			R3.Reamer[1](
				(*FB Inputs*)
					Enable_Motion:= All_Estops_OK,
					Fronius_Ream:= TRUE,
                    Binzel_Ream:= FALSE,  (*optional*)
					
					Ream_REQ:= R3.Peripheral_Req.1 AND ((R3.Task_ID_Ack=Tip_Dress)OR (R3.In_T1 AND R3.Peripheral_Req.5)),
					Ream_Time:= T#2S,
					Ream_Clamp_Open:= R3.Reamer[1].N01.I.1,
					Spray_REQ:= R3.Peripheral_Req.2 AND ((R3.Task_ID_Ack=Tip_Dress)OR (R3.In_T1 AND R3.Peripheral_Req.5)),
					Spray_Time:= T#2S,
					F_WireCutter_REQ:= R3.Peripheral_Req.4 AND ((R3.Task_ID_Ack=Tip_Dress)OR (R3.In_T1 AND R3.Peripheral_Req.5)),
					F_WireCutter_Time:= T#1S,
					
				(*FB Outputs*)
					Reaming_Complete=> ,(*mapped in cell services*)
					(*The following are for Binzel type reamers only*)
					LifterUp_ACK=> , (*mapped in cell services*)
					Clamp_ACK=>,(*mapped in cell services*)
					Injector_ACK=> ,(*mapped in cell services*)
					WireCutter_ACK=> (*mapped in cell services*)
					);
			
			(*R3.Reamer[1](
				(*FB Inputs*)
					Enable_Motion:= All_Estops_OK,
					Fronius_Ream:= TRUE,
                    Binzel_Ream:= FALSE,  (*optional*)
					Ream_REQ:= R3.Peripheral_Req.5 AND (R3.Task_ID_Ack=Tip_Dress),

				(*FB Outputs*)
					Reaming_Complete=> ,(*mapped in cell services*)
					);*)
		(*Call Actual Object*)
		R3();
		(*Output Data*)
		Out_To_ICxx.Robot[3].Robot_Type:= R3.FB_In.Robot_Type;
		Out_To_ICxx.Robot[3].Status:= R3.Status;
		Out_To_ICxx.Robot[3].Axis_Data[1]:= R3.S_Axis_Pos_Raw;
		Out_To_ICxx.Robot[3].In_Image:= R3.Input_Image;
		Out_To_ICxx.Robot[3].Out_Image:= R3.Output_Image;
		Out_To_ICxx.Robot[3].Discrete_ImageFSOE:= R3.Discrete_Image_FSoE;
		Out_To_ICxx.Robot[3].Options:= R3.FB_In.Options;
			Out_To_ICxx.Robot[3].WS_Discrete_Image[1]:= R3.WS[1].Discrete_Image;
			Out_To_ICxx.Robot[3].WS_Discrete_Image[2]:= R3.WS[2].Discrete_Image;
 			Out_To_ICxx.Robot[3].ATI_Discrete_Image:= R3.ATI[1].Discrete_Image;
			Out_To_ICxx.Robot[3].Reamer_Discrete_Image:= R3.Reamer[1].Discrete_Image;
			Out_To_ICxx.Robot[3].Fronius_Status:= R3.Fronius_Status;
		Out_To_ICxx.Robot[3].Ped_IO_ToShow[1]:= 0;			(*Set to Ped value if this robots ecat string contains the Ped's IO*)
		Out_To_ICxx.Robot[3].Ped_IO_ToShow[2]:= 0;			(*Set to Ped value if this robots ecat string contains the Ped's IO*)
		Out_To_ICxx.Robot[3].ECAT_Cable_Breaks:= R3.ECatSlave_Cable_Breaks;
		Out_To_ICxx.Robot[3].CT:= R3.CT;


(*R4 ------------------------*)
		(*Input Data*)
		R4.FB_In.Robot_Type:=KUKA_KRC4_SAFEOP;
		R4.FB_In.Install_Zero_Orientation:= 0; 	(*Set this value between 0 and 359 to set the zero position of the robot physical install with reference to 12 o'clock symbol on UI screens*)
		R4.FB_In.Under_Construction:= GTAC_CONFIG.Under_Construction;
		R4.FB_In.In_SIM_Mode:= GTAC_CONFIG.In_SIM_Mode;
		R4.FB_In.SIM_StartWorkAround:= FALSE;  (*Main.SIM_WorkAround_StartRobots*)
		R4.FB_In.CoE_Read_Trigger:= (GTAC_CONFIG.Option_Robot_Count>=4) AND Pulse_CoERead;
		R4.FB_In.Ecat_Master_AmsNetID:= MAIN.ECAT_Master.AmsID;
		R4.FB_In.Prev_EcatNode_Present:= NOT R3.EK1100_NotPresent; (*Ensure Previous Node Exists to determine Ecat Cable Break of this Devices Input Cable*)
		R4.FB_In.Safety_RST:=SAFETY_RESET;
		R4.FB_In.Enable_Motion:= All_Estops_OK OR GTAC_CONFIG.Under_Construction;
		R4.FB_In.Alarm_RST:=In_From_ICxx.ControlPower1;
		R4.FB_In.Select_Play:=FALSE;
		R4.FB_In.Select_Teach:=FALSE;
		R4.FB_In.Select_Remote:=FALSE;
		R4.FB_In.Start_Scan:=In_From_ICxx.StartRobots;
		R4.FB_In.Stop_Scan:=In_From_ICxx.StopRobots;
		R4.FB_In.Stop_Scan2:=FALSE;
		R4.FB_In.In_DryCycle:= GTAC_CONFIG.Dry_Cycle_Enabled;
		R4.FB_In.Low_Speed:= GTAC_CONFIG.Low_Speed_Enabled;
		R4.FB_In.Speed_Request:= In_From_ICxx.Global_Robot_Speed;
		R4.FB_In.Force_MasterTest_Req:= Cell_Services_Prog.Human_Reqs_MasterTest OR Cell_Services_Prog.A_Robot_Reqs_MasterTest;
		R4.FB_In.Force_BrakeTest_Req:= Cell_Services_Prog.Human_Reqs_BrakeTest OR Cell_Services_Prog.A_Robot_Reqs_BrakeTest;
		R4.FB_In.Major_Faults:= Faults.System_Major_Fault;
		R4.FB_In.Teach_Interlock:=R4_Data.Teach_Interlock;
		R4.FB_In.Weld_Inhibit:=In_From_ICxx.Rxx_Weld_Inhibit;
		R4.FB_In.Option_Disable_WaterFLT:= FALSE AND GTAC_CONFIG.Under_Construction OR (MAIN.R4.Task_ID_Ack=Tip_Change_EXT); (*Used to disable water fault if no water is present. use with caution*)
		R4.FB_In.OK_ToEnter_EquipInterf1:=R4_Data.OK_ToEnter_EquipInterf1;
		R4.FB_In.OK_ToEnter_EquipInterf2:=R4_Data.OK_ToEnter_EquipInterf2;
		R4.FB_In.OK_ToEnter_EquipInterf3:=R4_Data.OK_ToEnter_EquipInterf3;
		R4.FB_In.OK_ToEnter_EquipInterf4:=R4_Data.OK_ToEnter_EquipInterf4;
		R4.FB_In.OK_ToEnter_EquipInterf5:=R4_Data.OK_ToEnter_EquipInterf5;
		R4.FB_In.OK_ToEnter_EquipInterf6:=R4_Data.OK_ToEnter_EquipInterf6;
		R4.FB_In.OK_ToEnter_EquipInterf7:=R4_Data.OK_ToEnter_EquipInterf7;
		R4.FB_In.OK_ToEnter_EquipInterf8:=R4_Data.OK_ToEnter_EquipInterf8;
		R4.FB_In.OK_ToEnter_EquipInterf9:=R4_Data.OK_ToEnter_EquipInterf9;
		R4.FB_In.OK_ToEnter_HumanInterf1:=R4_Data.OK_ToEnter_HumanInterf1;
		R4.FB_In.OK_ToEnter_HumanInterf2:=R4_Data.OK_ToEnter_HumanInterf2;
		R4.FB_In.OK_ToEnter_HumanInterf3:=R4_Data.OK_ToEnter_HumanInterf3;
		R4.FB_In.OK_ToEnter_HumanInterf4:=R4_Data.OK_ToEnter_HumanInterf4;
		R4.FB_In.OK_ToEnter_HumanInterf5:=R4_Data.OK_ToEnter_HumanInterf5;
		R4.FB_In.OK_ToEnter_HumanInterf6:=R4_Data.OK_ToEnter_HumanInterf6;
		R4.FB_In.OK_ToEnter_HumanInterf7:=R4_Data.OK_ToEnter_HumanInterf7;
		R4.FB_In.OK_ToEnter_RobotInterfs:= R4_Data.OK_ToEnter_RobotInterfs;
		R4.FB_In.Fix_ID:=R4_Data.Fix_ID[R4.Location_Index];
		R4.FB_In.Model_ID:=R4_Data.Model_ID[R4.Location_Index];
		R4.FB_In.Task_ID:=R4_Data.Task_ID[R4.Location_Index];
		R4.FB_In.Proceed_From_Pounce:=R4_Data.Proceed_From_Pounce[R4.Location_Index];
		R4.FB_In.Complete_Ack:=R4_Data.Complete_Ack[R4.Location_Index];
		R4.FB_In.PeripheralReq_Ack:=R4_Data.PeripheralReq_Ack[R4.Location_Index];
		R4.FB_In.AuxReq_Ack:=R4_Data.AuxReq_Ack[R4.Location_Index];
		R4.FB_In.User_Inputs.0:= FALSE;
		R4.FB_In.User_Inputs.1:= FALSE;
		R4.FB_In.User_Inputs.2:= FALSE;
		R4.FB_In.User_Inputs.3:= FALSE;
		R4.FB_In.User_Inputs.4:= FALSE;
		R4.FB_In.User_Inputs.5:= FALSE;
		R4.FB_In.User_Inputs.6:= FALSE;
		R4.FB_In.User_Inputs.7:= FALSE;
			(*Configure Options Amounts*)
			R4.FB_In.Options.WeldCont_Amount:=0; 					(*Select amount of Spot Type Weld Controllers here (0 min, 4 max)*)
			R4.FB_In.Options.WaterStand_Amount:= 0;				(*Select amount of Water Stands here (0 min, 2 max)*)
			R4.FB_In.Options.MIGCont_Amount:= 0;					(*Select amount of MIG Type Weld Controllers here (0 min, 1 max)*)
			R4.FB_In.Options.Reamer_Amount:= 0;					(*Select amount of Tip Reamers here (0 min, 1 max)*)
			R4.FB_In.Options.EOAT_Amount:= 1;						(*Assign EOAT number to robot (0 min, 10 max)*)
			(*Configure Options Parameters*)

		(*Call Actual Object*)
		R4();
		(*Output Data*)
		Out_To_ICxx.Robot[4].Robot_Type:= R4.FB_In.Robot_Type;
		Out_To_ICxx.Robot[4].Status:= R4.Status;
		Out_To_ICxx.Robot[4].Axis_Data[1]:= R4.S_Axis_Pos_Raw;
		Out_To_ICxx.Robot[4].Axis_Data[7]:= R4.External_Axis_Pos_Raw; (*Actual value coming from robot*)
		Out_To_ICxx.Robot[4].In_Image:= R4.Input_Image;
		Out_To_ICxx.Robot[4].Out_Image:= R4.Output_Image;
		Out_To_ICxx.Robot[4].Discrete_ImageFSOE:= R4.Discrete_Image_FSoE;
		Out_To_ICxx.Robot[4].Options:= R4.FB_In.Options;
			Out_To_ICxx.Robot[4].WS_Discrete_Image[1]:= R4.WS[1].Discrete_Image;
			Out_To_ICxx.Robot[4].WS_Discrete_Image[2]:= R4.WS[2].Discrete_Image;
 			Out_To_ICxx.Robot[4].ATI_Discrete_Image:= R4.ATI[1].Discrete_Image;
			Out_To_ICxx.Robot[4].Reamer_Discrete_Image:= R4.Reamer[1].Discrete_Image;
			Out_To_ICxx.Robot[4].Fronius_Status:= R4.Fronius_Status;
		Out_To_ICxx.Robot[4].Ped_IO_ToShow[1]:= 0;			(*Set to Ped value if this robots ecat string contains the Ped's IO*)
		Out_To_ICxx.Robot[4].Ped_IO_ToShow[2]:= 0;			(*Set to Ped value if this robots ecat string contains the Ped's IO*)
		Out_To_ICxx.Robot[4].ECAT_Cable_Breaks:= R4.ECatSlave_Cable_Breaks;
		Out_To_ICxx.Robot[4].CT:= R4.CT;



(*R5 ------------------------*)
		(*Input Data*)
		R5.FB_In.Robot_Type:=KUKA_KRC4_SAFEOP_Turntable;
		R5.FB_In.Install_Zero_Orientation:= 0; 	(*Set this value between 0 and 359 to set the zero position of the robot physical install with reference to 12 o'clock symbol on UI screens*)
		R5.FB_In.Under_Construction:= GTAC_CONFIG.Under_Construction;
		R5.FB_In.In_SIM_Mode:= GTAC_CONFIG.In_SIM_Mode;
		R5.FB_In.SIM_StartWorkAround:= FALSE;  (*Main.SIM_WorkAround_StartRobots*)
		R5.FB_In.CoE_Read_Trigger:= (GTAC_CONFIG.Option_Robot_Count>=5) AND Pulse_CoERead;
		R5.FB_In.Ecat_Master_AmsNetID:= MAIN.ECAT_Master.AmsID;
		R5.FB_In.Prev_EcatNode_Present:= NOT R4.EK1100_NotPresent; (*Ensure Previous Node Exists to determine Ecat Cable Break of this Devices Input Cable*)
		R5.FB_In.Safety_RST:=SAFETY_RESET;
		R5.FB_In.Enable_Motion:= All_Estops_OK OR GTAC_CONFIG.Under_Construction;
		R5.FB_In.Alarm_RST:=In_From_ICxx.ControlPower1;
		R5.FB_In.Select_Play:=FALSE;
		R5.FB_In.Select_Teach:=FALSE;
		R5.FB_In.Select_Remote:=FALSE;
		R5.FB_In.Start_Scan:=In_From_ICxx.StartRobots;
		R5.FB_In.Stop_Scan:=In_From_ICxx.StopRobots;
		R5.FB_In.Stop_Scan2:=FALSE;
		R5.FB_In.In_DryCycle:= GTAC_CONFIG.Dry_Cycle_Enabled;
		R5.FB_In.Low_Speed:= GTAC_CONFIG.Low_Speed_Enabled;
		R5.FB_In.Speed_Request:= In_From_ICxx.Global_Robot_Speed;
		R5.FB_In.Force_MasterTest_Req:= Cell_Services_Prog.Human_Reqs_MasterTest OR Cell_Services_Prog.A_Robot_Reqs_MasterTest;
		R5.FB_In.Force_BrakeTest_Req:= Cell_Services_Prog.Human_Reqs_BrakeTest OR Cell_Services_Prog.A_Robot_Reqs_BrakeTest;
		R5.FB_In.Major_Faults:= Faults.System_Major_Fault;
		R5.FB_In.Teach_Interlock:=R5_Data.Teach_Interlock;
		R5.FB_In.Weld_Inhibit:=In_From_ICxx.Rxx_Weld_Inhibit;
		R5.FB_In.Option_Disable_WaterFLT:= FALSE AND GTAC_CONFIG.Under_Construction OR (MAIN.R5.Task_ID_Ack=Tip_Change_EXT); (*Used to disable water fault if no water is present. use with caution*)
		R5.FB_In.OK_ToEnter_EquipInterf1:=R5_Data.OK_ToEnter_EquipInterf1;
		R5.FB_In.OK_ToEnter_EquipInterf2:=R5_Data.OK_ToEnter_EquipInterf2;
		R5.FB_In.OK_ToEnter_EquipInterf3:=R5_Data.OK_ToEnter_EquipInterf3;
		R5.FB_In.OK_ToEnter_EquipInterf4:=R5_Data.OK_ToEnter_EquipInterf4;
		R5.FB_In.OK_ToEnter_EquipInterf5:=R5_Data.OK_ToEnter_EquipInterf5;
		R5.FB_In.OK_ToEnter_EquipInterf6:=R5_Data.OK_ToEnter_EquipInterf6;
		R5.FB_In.OK_ToEnter_EquipInterf7:=R5_Data.OK_ToEnter_EquipInterf7;
		R5.FB_In.OK_ToEnter_EquipInterf8:=R5_Data.OK_ToEnter_EquipInterf8;
		R5.FB_In.OK_ToEnter_EquipInterf9:=R5_Data.OK_ToEnter_EquipInterf9;
		R5.FB_In.OK_ToEnter_HumanInterf1:=R5_Data.OK_ToEnter_HumanInterf1;
		R5.FB_In.OK_ToEnter_HumanInterf2:=R5_Data.OK_ToEnter_HumanInterf2;
		R5.FB_In.OK_ToEnter_HumanInterf3:=R5_Data.OK_ToEnter_HumanInterf3;
		R5.FB_In.OK_ToEnter_HumanInterf4:=R5_Data.OK_ToEnter_HumanInterf4;
		R5.FB_In.OK_ToEnter_HumanInterf5:=R5_Data.OK_ToEnter_HumanInterf5;
		R5.FB_In.OK_ToEnter_HumanInterf6:=R5_Data.OK_ToEnter_HumanInterf6;
		R5.FB_In.OK_ToEnter_HumanInterf7:=R5_Data.OK_ToEnter_HumanInterf7;
		R5.FB_In.OK_ToEnter_HumanInterf8:=R5_Data.OK_ToEnter_HumanInterf8;
		R5.FB_In.OK_ToEnter_RobotInterfs:= R5_Data.OK_ToEnter_RobotInterfs;
		R5.FB_In.Fix_ID:=R5_Data.Fix_ID[R5.Location_Index];
		R5.FB_In.Model_ID:=R5_Data.Model_ID[R5.Location_Index];
		R5.FB_In.Task_ID:=R5_Data.Task_ID[R5.Location_Index];
		R5.FB_In.Proceed_From_Pounce:=R5_Data.Proceed_From_Pounce[R5.Location_Index];
		R5.FB_In.Complete_Ack:=R5_Data.Complete_Ack[R5.Location_Index];
		R5.FB_In.PeripheralReq_Ack:=R5_Data.PeripheralReq_Ack[R5.Location_Index];
		R5.FB_In.AuxReq_Ack:=R5_Data.AuxReq_Ack[R5.Location_Index];
		R5.FB_In.User_Inputs.0:= FALSE;
		R5.FB_In.User_Inputs.1:= FALSE;
		R5.FB_In.User_Inputs.2:= FALSE;
		R5.FB_In.User_Inputs.3:= FALSE;
		R5.FB_In.User_Inputs.4:= FALSE;
		R5.FB_In.User_Inputs.5:= FALSE;
		R5.FB_In.User_Inputs.6:= FALSE;
		R5.FB_In.User_Inputs.7:= FALSE;
			(*Configure Options Amounts*)
			R5.FB_In.Options.WeldCont_Amount:= 0; 					(*Select amount of Spot Type Weld Controllers here (0 min, 4 max)*)
			R5.FB_In.Options.WaterStand_Amount:= 0;				(*Select amount of Water Stands here (0 min, 2 max)*)
			R5.FB_In.Options.MIGCont_Amount:= 1;					(*Select amount of MIG Type Weld Controllers here (0 min, 1 max)*)
			R5.FB_In.Options.Reamer_Amount:= 1;					(*Select amount of Tip Reamers here (0 min, 1 max)*)
			R5.FB_In.Options.EOAT_Amount:= 0;						(*Assign EOAT number to robot (0 min, 10 max)*)
			(*Configure Options Parameters*)
			
			R5.Reamer[1](
				(*FB Inputs*)
					Enable_Motion:= All_Estops_OK,
					Fronius_Ream:= TRUE,
                    Binzel_Ream:= FALSE,  (*optional*)
					
					Ream_REQ:= R5.Peripheral_Req.1 AND ((R5.Task_ID_Ack=Tip_Dress)OR (R5.In_T1 AND R5.Peripheral_Req.5)),
					Ream_Time:= T#2S,
					Ream_Clamp_Open:= R5.Reamer[1].N01.I.1,
					Spray_REQ:= R5.Peripheral_Req.2 AND ((R5.Task_ID_Ack=Tip_Dress)OR (R5.In_T1 AND R5.Peripheral_Req.5)),
					Spray_Time:= T#2S,
					F_WireCutter_REQ:= R5.Peripheral_Req.4 AND ((R5.Task_ID_Ack=Tip_Dress)OR (R5.In_T1 AND R5.Peripheral_Req.5)),
					F_WireCutter_Time:= T#1S,
					
				(*FB Outputs*)
					Reaming_Complete=> ,(*mapped in cell services*)
					(*The following are for Binzel type reamers only*)
					LifterUp_ACK=> , (*mapped in cell services*)
					Clamp_ACK=>,(*mapped in cell services*)
					Injector_ACK=> ,(*mapped in cell services*)
					WireCutter_ACK=> (*mapped in cell services*)
					);
			(*R5.Reamer[1](
				(*FB Inputs*)
					Enable_Motion:= All_Estops_OK,
					Fronius_Ream:= TRUE,
                    Binzel_Ream:= FALSE,  (*optional*)
					Ream_REQ:= R5.Peripheral_Req.5 AND (R5.Task_ID_Ack=Tip_Dress),

				(*FB Outputs*)
					Reaming_Complete=> ,(*mapped in cell services*)
					);*)
		(*Call Actual Object*)
		R5();
		(*Output Data*)
		Out_To_ICxx.Robot[5].Robot_Type:= R5.FB_In.Robot_Type;
		Out_To_ICxx.Robot[5].Status:= R5.Status;
		Out_To_ICxx.Robot[5].Axis_Data[1]:= R5.S_Axis_Pos_Raw;
		Out_To_ICxx.Robot[5].In_Image:= R5.Input_Image;
		Out_To_ICxx.Robot[5].Out_Image:= R5.Output_Image;
		Out_To_ICxx.Robot[5].Discrete_ImageFSOE:= R5.Discrete_Image_FSoE;
		Out_To_ICxx.Robot[5].Options:= R5.FB_In.Options;
			Out_To_ICxx.Robot[5].WS_Discrete_Image[1]:= R5.WS[1].Discrete_Image;
			Out_To_ICxx.Robot[5].WS_Discrete_Image[2]:= R5.WS[2].Discrete_Image;
 			Out_To_ICxx.Robot[5].ATI_Discrete_Image:= R5.ATI[1].Discrete_Image;
			Out_To_ICxx.Robot[5].Reamer_Discrete_Image:= R5.Reamer[1].Discrete_Image;
			Out_To_ICxx.Robot[5].Fronius_Status:= R5.Fronius_Status;
		Out_To_ICxx.Robot[5].Ped_IO_ToShow[1]:= 0;			(*Set to Ped value if this robots ecat string contains the Ped's IO*)
		Out_To_ICxx.Robot[5].Ped_IO_ToShow[2]:= 0;			(*Set to Ped value if this robots ecat string contains the Ped's IO*)
		Out_To_ICxx.Robot[5].ECAT_Cable_Breaks:= R5.ECatSlave_Cable_Breaks;
		Out_To_ICxx.Robot[5].CT:= R5.CT;
		(*Example of passing Turntable Axis Data*)
		//Out_To_ICxx.TT02_Location_Index:= R5.TT_Axis_Location_Index; (*Pass Turntable location*) DEBUG - RESTORE AFTER SIM - RJ
		
		(*IF (MAIN.SIM_WorkAround_TT02_Position_Index[0] = TRUE)
			THEN Out_To_ICxx.TT02_Location_Index:= 1;
		ELSIF (MAIN.SIM_WorkAround_TT02_Position_Index[1] = TRUE)
			THEN Out_To_ICxx.TT02_Location_Index:= 2;
		ELSE
			Out_To_ICxx.TT02_Location_Index:= 0;
		END_IF*)	//DEBUG - RJ - REMOVE ABOVE AFTER SIM, RESTORE original Out_To_ICxx.TT01_Location_Index:= R1.TT_Axis_Location_Index;
		Out_To_ICxx.TT02_Location_Index:= R5.TT_Axis_Location_Index;



(*R6 ------------------------*)
		(*Input Data*)
		R6.FB_In.Robot_Type:=KUKA_KRC4_SAFEOP;
		R6.FB_In.Install_Zero_Orientation:= 0; 	(*Set this value between 0 and 359 to set the zero position of the robot physical install with reference to 12 o'clock symbol on UI screens*)
		R6.FB_In.Under_Construction:= GTAC_CONFIG.Under_Construction;
		R6.FB_In.In_SIM_Mode:= GTAC_CONFIG.In_SIM_Mode;
		R6.FB_In.SIM_StartWorkAround:= FALSE;  (*Main.SIM_WorkAround_StartRobots*)
		R6.FB_In.CoE_Read_Trigger:= (GTAC_CONFIG.Option_Robot_Count>=6) AND Pulse_CoERead;
		R6.FB_In.Ecat_Master_AmsNetID:= MAIN.ECAT_Master.AmsID;
		R6.FB_In.Prev_EcatNode_Present:= NOT R5.EK1100_NotPresent; (*Ensure Previous Node Exists to determine Ecat Cable Break of this Devices Input Cable*)
		R6.FB_In.Safety_RST:=SAFETY_RESET;
		R6.FB_In.Enable_Motion:= All_Estops_OK OR GTAC_CONFIG.Under_Construction;
		R6.FB_In.Alarm_RST:=In_From_ICxx.ControlPower1;
		R6.FB_In.Select_Play:=FALSE;
		R6.FB_In.Select_Teach:=FALSE;
		R6.FB_In.Select_Remote:=FALSE;
		R6.FB_In.Start_Scan:=In_From_ICxx.StartRobots;
		R6.FB_In.Stop_Scan:=In_From_ICxx.StopRobots;
		R6.FB_In.Stop_Scan2:=FALSE;
		R6.FB_In.In_DryCycle:= GTAC_CONFIG.Dry_Cycle_Enabled;
		R6.FB_In.Low_Speed:= GTAC_CONFIG.Low_Speed_Enabled;
		R6.FB_In.Speed_Request:= In_From_ICxx.Global_Robot_Speed;
		R6.FB_In.Force_MasterTest_Req:= Cell_Services_Prog.Human_Reqs_MasterTest OR Cell_Services_Prog.A_Robot_Reqs_MasterTest;
		R6.FB_In.Force_BrakeTest_Req:= Cell_Services_Prog.Human_Reqs_BrakeTest OR Cell_Services_Prog.A_Robot_Reqs_BrakeTest;
		R6.FB_In.Major_Faults:= Faults.System_Major_Fault;
		R6.FB_In.Teach_Interlock:=R6_Data.Teach_Interlock;
		R6.FB_In.Weld_Inhibit:=In_From_ICxx.Rxx_Weld_Inhibit;
		R6.FB_In.Option_Disable_WaterFLT:= FALSE AND GTAC_CONFIG.Under_Construction OR (MAIN.R6.Task_ID_Ack=Tip_Change_EXT); (*Used to disable water fault if no water is present. use with caution*)
		R6.FB_In.OK_ToEnter_EquipInterf1:=R6_Data.OK_ToEnter_EquipInterf1;
		R6.FB_In.OK_ToEnter_EquipInterf2:=R6_Data.OK_ToEnter_EquipInterf2;
		R6.FB_In.OK_ToEnter_EquipInterf3:=R6_Data.OK_ToEnter_EquipInterf3;
		R6.FB_In.OK_ToEnter_EquipInterf4:=R6_Data.OK_ToEnter_EquipInterf4;
		R6.FB_In.OK_ToEnter_EquipInterf5:=R6_Data.OK_ToEnter_EquipInterf5;
		R6.FB_In.OK_ToEnter_EquipInterf6:=R6_Data.OK_ToEnter_EquipInterf6;
		R6.FB_In.OK_ToEnter_EquipInterf7:=R6_Data.OK_ToEnter_EquipInterf7;
		R6.FB_In.OK_ToEnter_EquipInterf8:=R6_Data.OK_ToEnter_EquipInterf8;
		R6.FB_In.OK_ToEnter_EquipInterf9:=R6_Data.OK_ToEnter_EquipInterf9;
		R6.FB_In.OK_ToEnter_HumanInterf1:=R6_Data.OK_ToEnter_HumanInterf1;
		R6.FB_In.OK_ToEnter_HumanInterf2:=R6_Data.OK_ToEnter_HumanInterf2;
		R6.FB_In.OK_ToEnter_HumanInterf3:=R6_Data.OK_ToEnter_HumanInterf3;
		R6.FB_In.OK_ToEnter_HumanInterf4:=R6_Data.OK_ToEnter_HumanInterf4;
		R6.FB_In.OK_ToEnter_HumanInterf5:=R6_Data.OK_ToEnter_HumanInterf5;
		R6.FB_In.OK_ToEnter_HumanInterf6:=R6_Data.OK_ToEnter_HumanInterf6;
		R6.FB_In.OK_ToEnter_HumanInterf7:=R6_Data.OK_ToEnter_HumanInterf7;
		R6.FB_In.OK_ToEnter_HumanInterf8:=R6_Data.OK_ToEnter_HumanInterf8;
		R6.FB_In.OK_ToEnter_RobotInterfs:= R6_Data.OK_ToEnter_RobotInterfs;
		R6.FB_In.Fix_ID:=R6_Data.Fix_ID[R6.Location_Index];
		R6.FB_In.Model_ID:=R6_Data.Model_ID[R6.Location_Index];
		R6.FB_In.Task_ID:=R6_Data.Task_ID[R6.Location_Index];
		R6.FB_In.Proceed_From_Pounce:=R6_Data.Proceed_From_Pounce[R6.Location_Index];
		R6.FB_In.Complete_Ack:=R6_Data.Complete_Ack[R6.Location_Index];
		R6.FB_In.PeripheralReq_Ack:=R6_Data.PeripheralReq_Ack[R6.Location_Index];
		R6.FB_In.AuxReq_Ack:=R6_Data.AuxReq_Ack[R6.Location_Index];
		R6.FB_In.User_Inputs.0:= FALSE;
		R6.FB_In.User_Inputs.1:= FALSE;
		R6.FB_In.User_Inputs.2:= FALSE;
		R6.FB_In.User_Inputs.3:= FALSE;
		R6.FB_In.User_Inputs.4:= FALSE;
		R6.FB_In.User_Inputs.5:= FALSE;
		R6.FB_In.User_Inputs.6:= FALSE;
		R6.FB_In.User_Inputs.7:= FALSE;
			(*Configure Options Amounts*)
			R6.FB_In.Options.WeldCont_Amount:= 0; 					(*Select amount of Spot Type Weld Controllers here (0 min, 4 max)*)
			R6.FB_In.Options.WaterStand_Amount:= 0;				(*Select amount of Water Stands here (0 min, 2 max)*)
			R6.FB_In.Options.MIGCont_Amount:= 1;					(*Select amount of MIG Type Weld Controllers here (0 min, 1 max)*)
			R6.FB_In.Options.Reamer_Amount:= 1;					(*Select amount of Tip Reamers here (0 min, 1 max)*)
			R6.FB_In.Options.EOAT_Amount:= 0;						(*Assign EOAT number to robot (0 min, 10 max)*)
			(*Configure Options Parameters*)
			
			R6.Reamer[1](
				(*FB Inputs*)
					Enable_Motion:= All_Estops_OK,
					Fronius_Ream:= TRUE,
                    Binzel_Ream:= FALSE,  (*optional*)
					
					Ream_REQ:= R6.Peripheral_Req.1 AND ((R6.Task_ID_Ack=Tip_Dress)OR (R6.In_T1 AND R6.Peripheral_Req.5)),
					Ream_Time:= T#2S,
					Ream_Clamp_Open:= R6.Reamer[1].N01.I.1,
					Spray_REQ:= R6.Peripheral_Req.2 AND ((R6.Task_ID_Ack=Tip_Dress)OR (R6.In_T1 AND R6.Peripheral_Req.5)),
					Spray_Time:= T#2S,
					F_WireCutter_REQ:= R6.Peripheral_Req.4 AND ((R6.Task_ID_Ack=Tip_Dress)OR (R6.In_T1 AND R6.Peripheral_Req.5)),
					F_WireCutter_Time:= T#1S,
					
				(*FB Outputs*)
					Reaming_Complete=> ,(*mapped in cell services*)
					(*The following are for Binzel type reamers only*)
					LifterUp_ACK=> , (*mapped in cell services*)
					Clamp_ACK=>,(*mapped in cell services*)
					Injector_ACK=> ,(*mapped in cell services*)
					WireCutter_ACK=> (*mapped in cell services*)
					);
			(*R6.Reamer[1](
				(*FB Inputs*)
					Enable_Motion:= All_Estops_OK,
					Fronius_Ream:= TRUE,
                    Binzel_Ream:= FALSE,  (*optional*)
					Ream_REQ:= R6.Peripheral_Req.5 AND (R6.Task_ID_Ack=Tip_Dress),

				(*FB Outputs*)
					Reaming_Complete=> ,(*mapped in cell services*)
					);*)
		(*Call Actual Object*)
		R6();
		(*Output Data*)
		Out_To_ICxx.Robot[6].Robot_Type:= R6.FB_In.Robot_Type;
		Out_To_ICxx.Robot[6].Status:= R6.Status;
		Out_To_ICxx.Robot[6].Axis_Data[1]:= R6.S_Axis_Pos_Raw;
		Out_To_ICxx.Robot[6].In_Image:= R6.Input_Image;
		Out_To_ICxx.Robot[6].Out_Image:= R6.Output_Image;
		Out_To_ICxx.Robot[6].Discrete_ImageFSOE:= R6.Discrete_Image_FSoE;
		Out_To_ICxx.Robot[6].Options:= R6.FB_In.Options;
			Out_To_ICxx.Robot[6].WS_Discrete_Image[1]:= R6.WS[1].Discrete_Image;
			Out_To_ICxx.Robot[6].WS_Discrete_Image[2]:= R6.WS[2].Discrete_Image;
 			Out_To_ICxx.Robot[6].ATI_Discrete_Image:= R6.ATI[1].Discrete_Image;
			Out_To_ICxx.Robot[6].Reamer_Discrete_Image:= R6.Reamer[1].Discrete_Image;
			Out_To_ICxx.Robot[6].Fronius_Status:= R6.Fronius_Status;
		Out_To_ICxx.Robot[6].Ped_IO_ToShow[1]:= 0;			(*Set to Ped value if this robots ecat string contains the Ped's IO*)
		Out_To_ICxx.Robot[6].Ped_IO_ToShow[2]:= 0;			(*Set to Ped value if this robots ecat string contains the Ped's IO*)
		Out_To_ICxx.Robot[6].ECAT_Cable_Breaks:= R6.ECatSlave_Cable_Breaks;
		Out_To_ICxx.Robot[6].CT:= R6.CT;



(*R7 ------------------------*)
		(*Input Data*)
		R7.FB_In.Robot_Type:=KUKA_KRC4_SAFEOP;
		R7.FB_In.Install_Zero_Orientation:= 0; 	(*Set this value between 0 and 359 to set the zero position of the robot physical install with reference to 12 o'clock symbol on UI screens*)
		R7.FB_In.Under_Construction:= GTAC_CONFIG.Under_Construction;
		R7.FB_In.In_SIM_Mode:= GTAC_CONFIG.In_SIM_Mode;
		R7.FB_In.SIM_StartWorkAround:= FALSE;  (*Main.SIM_WorkAround_StartRobots*)
		R7.FB_In.CoE_Read_Trigger:= (GTAC_CONFIG.Option_Robot_Count>=7) AND Pulse_CoERead;
		R7.FB_In.Ecat_Master_AmsNetID:= MAIN.ECAT_Master.AmsID;
		R7.FB_In.Prev_EcatNode_Present:= NOT R6.EK1100_NotPresent; (*Ensure Previous Node Exists to determine Ecat Cable Break of this Devices Input Cable*)
		R7.FB_In.Safety_RST:=SAFETY_RESET;
		R7.FB_In.Enable_Motion:= All_Estops_OK OR GTAC_CONFIG.Under_Construction;
		R7.FB_In.Alarm_RST:=In_From_ICxx.ControlPower1;
		R7.FB_In.Select_Play:=FALSE;
		R7.FB_In.Select_Teach:=FALSE;
		R7.FB_In.Select_Remote:=FALSE;
		R7.FB_In.Start_Scan:=In_From_ICxx.StartRobots;
		R7.FB_In.Stop_Scan:=In_From_ICxx.StopRobots;
		R7.FB_In.Stop_Scan2:=FALSE;
		R7.FB_In.In_DryCycle:= GTAC_CONFIG.Dry_Cycle_Enabled;
		R7.FB_In.Low_Speed:= GTAC_CONFIG.Low_Speed_Enabled;
		R7.FB_In.Speed_Request:= In_From_ICxx.Global_Robot_Speed;
		R7.FB_In.Force_MasterTest_Req:= Cell_Services_Prog.Human_Reqs_MasterTest OR Cell_Services_Prog.A_Robot_Reqs_MasterTest;
		R7.FB_In.Force_BrakeTest_Req:= Cell_Services_Prog.Human_Reqs_BrakeTest OR Cell_Services_Prog.A_Robot_Reqs_BrakeTest;
		R7.FB_In.Major_Faults:= Faults.System_Major_Fault;
		R7.FB_In.Teach_Interlock:=R7_Data.Teach_Interlock;
		R7.FB_In.Weld_Inhibit:=In_From_ICxx.Rxx_Weld_Inhibit;
		R7.FB_In.Option_Disable_WaterFLT:= FALSE AND GTAC_CONFIG.Under_Construction OR (MAIN.R7.Task_ID_Ack=Tip_Change_EXT); (*Used to disable water fault if no water is present. use with caution*)
		R7.FB_In.OK_ToEnter_EquipInterf1:=R7_Data.OK_ToEnter_EquipInterf1;
		R7.FB_In.OK_ToEnter_EquipInterf2:=R7_Data.OK_ToEnter_EquipInterf2;
		R7.FB_In.OK_ToEnter_EquipInterf3:=R7_Data.OK_ToEnter_EquipInterf3;
		R7.FB_In.OK_ToEnter_EquipInterf4:=R7_Data.OK_ToEnter_EquipInterf4;
		R7.FB_In.OK_ToEnter_EquipInterf5:=R7_Data.OK_ToEnter_EquipInterf5;
		R7.FB_In.OK_ToEnter_EquipInterf6:=R7_Data.OK_ToEnter_EquipInterf6;
		R7.FB_In.OK_ToEnter_EquipInterf7:=R7_Data.OK_ToEnter_EquipInterf7;
		R7.FB_In.OK_ToEnter_EquipInterf8:=R7_Data.OK_ToEnter_EquipInterf8;
		R7.FB_In.OK_ToEnter_EquipInterf9:=R7_Data.OK_ToEnter_EquipInterf9;
		R7.FB_In.OK_ToEnter_HumanInterf1:=R7_Data.OK_ToEnter_HumanInterf1;
		R7.FB_In.OK_ToEnter_HumanInterf2:=R7_Data.OK_ToEnter_HumanInterf2;
		R7.FB_In.OK_ToEnter_HumanInterf3:=R7_Data.OK_ToEnter_HumanInterf3;
		R7.FB_In.OK_ToEnter_HumanInterf4:=R7_Data.OK_ToEnter_HumanInterf4;
		R7.FB_In.OK_ToEnter_HumanInterf5:=R7_Data.OK_ToEnter_HumanInterf5;
		R7.FB_In.OK_ToEnter_HumanInterf6:=R7_Data.OK_ToEnter_HumanInterf6;
		R7.FB_In.OK_ToEnter_HumanInterf7:=R7_Data.OK_ToEnter_HumanInterf7;
		R7.FB_In.OK_ToEnter_HumanInterf8:=R7_Data.OK_ToEnter_HumanInterf8;
		R7.FB_In.OK_ToEnter_RobotInterfs:= R7_Data.OK_ToEnter_RobotInterfs;
		R7.FB_In.Fix_ID:=R7_Data.Fix_ID[R7.Location_Index];
		R7.FB_In.Model_ID:=R7_Data.Model_ID[R7.Location_Index];
		R7.FB_In.Task_ID:=R7_Data.Task_ID[R7.Location_Index];
		R7.FB_In.Proceed_From_Pounce:=R7_Data.Proceed_From_Pounce[R7.Location_Index];
		R7.FB_In.Complete_Ack:=R7_Data.Complete_Ack[R7.Location_Index];
		R7.FB_In.PeripheralReq_Ack:=R7_Data.PeripheralReq_Ack[R7.Location_Index];
		R7.FB_In.AuxReq_Ack:=R7_Data.AuxReq_Ack[R7.Location_Index];
		R7.FB_In.User_Inputs.0:= FALSE;
		R7.FB_In.User_Inputs.1:= FALSE;
		R7.FB_In.User_Inputs.2:= FALSE;
		R7.FB_In.User_Inputs.3:= FALSE;
		R7.FB_In.User_Inputs.4:= FALSE;
		R7.FB_In.User_Inputs.5:= FALSE;
		R7.FB_In.User_Inputs.6:= FALSE;
		R7.FB_In.User_Inputs.7:= FALSE;
			(*Configure Options Amounts*)
			R7.FB_In.Options.WeldCont_Amount:= 0; 					(*Select amount of Spot Type Weld Controllers here (0 min, 4 max)*)
			R7.FB_In.Options.WaterStand_Amount:= 0;				(*Select amount of Water Stands here (0 min, 2 max)*)
			R7.FB_In.Options.MIGCont_Amount:= 1;					(*Select amount of MIG Type Weld Controllers here (0 min, 1 max)*)
			R7.FB_In.Options.Reamer_Amount:= 1;					(*Select amount of Tip Reamers here (0 min, 1 max)*)
			R7.FB_In.Options.EOAT_Amount:= 0;						(*Assign EOAT number to robot (0 min, 10 max)*)
			(*Configure Options Parameters*)
			
			R7.Reamer[1](
				(*FB Inputs*)
					Enable_Motion:= All_Estops_OK,
					Fronius_Ream:= TRUE,
                    Binzel_Ream:= FALSE,  (*optional*)
					
					Ream_REQ:= R7.Peripheral_Req.1 AND ((R7.Task_ID_Ack=Tip_Dress)OR (R7.In_T1 AND R7.Peripheral_Req.5)),
					Ream_Time:= T#2S,
					Ream_Clamp_Open:= R7.Reamer[1].N01.I.1,
					Spray_REQ:= R7.Peripheral_Req.2 AND ((R7.Task_ID_Ack=Tip_Dress)OR (R7.In_T1 AND R7.Peripheral_Req.5)),
					Spray_Time:= T#2S,
					F_WireCutter_REQ:= R7.Peripheral_Req.4 AND ((R7.Task_ID_Ack=Tip_Dress)OR (R7.In_T1 AND R7.Peripheral_Req.5)),
					F_WireCutter_Time:= T#1S,
					
				(*FB Outputs*)
					Reaming_Complete=> ,(*mapped in cell services*)
					(*The following are for Binzel type reamers only*)
					LifterUp_ACK=> , (*mapped in cell services*)
					Clamp_ACK=>,(*mapped in cell services*)
					Injector_ACK=> ,(*mapped in cell services*)
					WireCutter_ACK=> (*mapped in cell services*)
					);
			(*R7.Reamer[1](
				(*FB Inputs*)
					Enable_Motion:= All_Estops_OK,
					Fronius_Ream:= TRUE,
                    Binzel_Ream:= FALSE,  (*optional*)
					Ream_REQ:= R7.Peripheral_Req.5 AND (R7.Task_ID_Ack=Tip_Dress),

				(*FB Outputs*)
					Reaming_Complete=> ,(*mapped in cell services*)
					);*)
		(*Call Actual Object*)
		R7();
		(*Output Data*)
		Out_To_ICxx.Robot[7].Robot_Type:= R7.FB_In.Robot_Type;
		Out_To_ICxx.Robot[7].Status:= R7.Status;
		Out_To_ICxx.Robot[7].Axis_Data[1]:= R7.S_Axis_Pos_Raw;
		Out_To_ICxx.Robot[7].In_Image:= R7.Input_Image;
		Out_To_ICxx.Robot[7].Out_Image:= R7.Output_Image;
		Out_To_ICxx.Robot[7].Discrete_ImageFSOE:= R7.Discrete_Image_FSoE;
		Out_To_ICxx.Robot[7].Options:= R7.FB_In.Options;
			Out_To_ICxx.Robot[7].WS_Discrete_Image[1]:= R7.WS[1].Discrete_Image;
			Out_To_ICxx.Robot[7].WS_Discrete_Image[2]:= R7.WS[2].Discrete_Image;
 			Out_To_ICxx.Robot[7].ATI_Discrete_Image:= R7.ATI[1].Discrete_Image;
			Out_To_ICxx.Robot[7].Reamer_Discrete_Image:= R7.Reamer[1].Discrete_Image;
			Out_To_ICxx.Robot[7].Fronius_Status:= R7.Fronius_Status;
		Out_To_ICxx.Robot[7].Ped_IO_ToShow[1]:= 0;			(*Set to Ped value if this robots ecat string contains the Ped's IO*)
		Out_To_ICxx.Robot[7].Ped_IO_ToShow[2]:= 0;			(*Set to Ped value if this robots ecat string contains the Ped's IO*)
		Out_To_ICxx.Robot[7].ECAT_Cable_Breaks:= R7.ECatSlave_Cable_Breaks;
		Out_To_ICxx.Robot[7].CT:= R7.CT;



(*R8 ------------------------*)
		(*Input Data*)
		R8.FB_In.Robot_Type:=KUKA_KRC4_SAFEOP;
		R8.FB_In.Install_Zero_Orientation:= 0; 	(*Set this value between 0 and 359 to set the zero position of the robot physical install with reference to 12 o'clock symbol on UI screens*)
		R8.FB_In.Under_Construction:= GTAC_CONFIG.Under_Construction;
		R8.FB_In.In_SIM_Mode:= GTAC_CONFIG.In_SIM_Mode;
		R8.FB_In.SIM_StartWorkAround:= FALSE;  (*Main.SIM_WorkAround_StartRobots*)
		R8.FB_In.CoE_Read_Trigger:= (GTAC_CONFIG.Option_Robot_Count>=8) AND Pulse_CoERead;
		R8.FB_In.Ecat_Master_AmsNetID:= MAIN.ECAT_Master.AmsID;
		R8.FB_In.Prev_EcatNode_Present:= NOT R7.EK1100_NotPresent; (*Ensure Previous Node Exists to determine Ecat Cable Break of this Devices Input Cable*)
		R8.FB_In.Safety_RST:=SAFETY_RESET;
		R8.FB_In.Enable_Motion:= All_Estops_OK OR GTAC_CONFIG.Under_Construction;
		R8.FB_In.Alarm_RST:=In_From_ICxx.ControlPower1;
		R8.FB_In.Select_Play:=FALSE;
		R8.FB_In.Select_Teach:=FALSE;
		R8.FB_In.Select_Remote:=FALSE;
		R8.FB_In.Start_Scan:=In_From_ICxx.StartRobots;
		R8.FB_In.Stop_Scan:=In_From_ICxx.StopRobots;
		R8.FB_In.Stop_Scan2:=FALSE;
		R8.FB_In.In_DryCycle:= GTAC_CONFIG.Dry_Cycle_Enabled;
		R8.FB_In.Low_Speed:= GTAC_CONFIG.Low_Speed_Enabled;
		R8.FB_In.Speed_Request:= In_From_ICxx.Global_Robot_Speed;
		R8.FB_In.Force_MasterTest_Req:= Cell_Services_Prog.Human_Reqs_MasterTest OR Cell_Services_Prog.A_Robot_Reqs_MasterTest;
		R8.FB_In.Force_BrakeTest_Req:= Cell_Services_Prog.Human_Reqs_BrakeTest OR Cell_Services_Prog.A_Robot_Reqs_BrakeTest;
		R8.FB_In.Major_Faults:= Faults.System_Major_Fault;
		R8.FB_In.Teach_Interlock:=R8_Data.Teach_Interlock;
		R8.FB_In.Weld_Inhibit:=In_From_ICxx.Rxx_Weld_Inhibit;
		R8.FB_In.Option_Disable_WaterFLT:= FALSE AND GTAC_CONFIG.Under_Construction OR (MAIN.R8.Task_ID_Ack=Tip_Change_EXT); (*Used to disable water fault if no water is present. use with caution*)
		R8.FB_In.OK_ToEnter_EquipInterf1:=R8_Data.OK_ToEnter_EquipInterf1;
		R8.FB_In.OK_ToEnter_EquipInterf2:=R8_Data.OK_ToEnter_EquipInterf2;
		R8.FB_In.OK_ToEnter_EquipInterf3:=R8_Data.OK_ToEnter_EquipInterf3;
		R8.FB_In.OK_ToEnter_EquipInterf4:=R8_Data.OK_ToEnter_EquipInterf4;
		R8.FB_In.OK_ToEnter_EquipInterf5:=R8_Data.OK_ToEnter_EquipInterf5;
		R8.FB_In.OK_ToEnter_EquipInterf6:=R8_Data.OK_ToEnter_EquipInterf6;
		R8.FB_In.OK_ToEnter_EquipInterf7:=R8_Data.OK_ToEnter_EquipInterf7;
		R8.FB_In.OK_ToEnter_EquipInterf8:=R8_Data.OK_ToEnter_EquipInterf8;
		R8.FB_In.OK_ToEnter_EquipInterf9:=R8_Data.OK_ToEnter_EquipInterf9;
		R8.FB_In.OK_ToEnter_HumanInterf1:=R8_Data.OK_ToEnter_HumanInterf1;
		R8.FB_In.OK_ToEnter_HumanInterf2:=R8_Data.OK_ToEnter_HumanInterf2;
		R8.FB_In.OK_ToEnter_HumanInterf3:=R8_Data.OK_ToEnter_HumanInterf3;
		R8.FB_In.OK_ToEnter_HumanInterf4:=R8_Data.OK_ToEnter_HumanInterf4;
		R8.FB_In.OK_ToEnter_HumanInterf5:=R8_Data.OK_ToEnter_HumanInterf5;
		R8.FB_In.OK_ToEnter_HumanInterf6:=R8_Data.OK_ToEnter_HumanInterf6;
		R8.FB_In.OK_ToEnter_HumanInterf7:=R8_Data.OK_ToEnter_HumanInterf7;
		R8.FB_In.OK_ToEnter_HumanInterf8:=R8_Data.OK_ToEnter_HumanInterf8;
		R8.FB_In.OK_ToEnter_RobotInterfs:= R8_Data.OK_ToEnter_RobotInterfs;
		R8.FB_In.Fix_ID:=R8_Data.Fix_ID[R8.Location_Index];
		R8.FB_In.Model_ID:=R8_Data.Model_ID[R8.Location_Index];
		R8.FB_In.Task_ID:=R8_Data.Task_ID[R8.Location_Index];
		R8.FB_In.Proceed_From_Pounce:=R8_Data.Proceed_From_Pounce[R8.Location_Index];
		R8.FB_In.Complete_Ack:=R8_Data.Complete_Ack[R8.Location_Index];
		R8.FB_In.PeripheralReq_Ack:=R8_Data.PeripheralReq_Ack[R8.Location_Index];
		R8.FB_In.AuxReq_Ack:=R8_Data.AuxReq_Ack[R8.Location_Index];
		R8.FB_In.User_Inputs.0:= FALSE;
		R8.FB_In.User_Inputs.1:= FALSE;
		R8.FB_In.User_Inputs.2:= FALSE;
		R8.FB_In.User_Inputs.3:= FALSE;
		R8.FB_In.User_Inputs.4:= FALSE;
		R8.FB_In.User_Inputs.5:= FALSE;
		R8.FB_In.User_Inputs.6:= FALSE;
		R8.FB_In.User_Inputs.7:= FALSE;
			(*Configure Options Amounts*)
			R8.FB_In.Options.WeldCont_Amount:= 0; 					(*Select amount of Spot Type Weld Controllers here (0 min, 4 max)*)
			R8.FB_In.Options.WaterStand_Amount:= 0;				(*Select amount of Water Stands here (0 min, 2 max)*)
			R8.FB_In.Options.MIGCont_Amount:= 1;					(*Select amount of MIG Type Weld Controllers here (0 min, 1 max)*)
			R8.FB_In.Options.Reamer_Amount:= 1;					(*Select amount of Tip Reamers here (0 min, 1 max)*)
			R8.FB_In.Options.EOAT_Amount:= 0;						(*Assign EOAT number to robot (0 min, 10 max)*)
			(*Configure Options Parameters*)
			
			R8.Reamer[1](
				(*FB Inputs*)
					Enable_Motion:= All_Estops_OK,
					Fronius_Ream:= TRUE,
                    Binzel_Ream:= FALSE,  (*optional*)
					
					Ream_REQ:= R8.Peripheral_Req.1 AND ((R8.Task_ID_Ack=Tip_Dress)OR (R8.In_T1 AND R8.Peripheral_Req.5)),
					Ream_Time:= T#2S,
					Ream_Clamp_Open:= R8.Reamer[1].N01.I.1,
					Spray_REQ:= R8.Peripheral_Req.2 AND ((R8.Task_ID_Ack=Tip_Dress)OR (R8.In_T1 AND R8.Peripheral_Req.5)),
					Spray_Time:= T#2S,
					F_WireCutter_REQ:= R8.Peripheral_Req.4 AND ((R8.Task_ID_Ack=Tip_Dress)OR (R8.In_T1 AND R8.Peripheral_Req.5)),
					F_WireCutter_Time:= T#1S,
					
				(*FB Outputs*)
					Reaming_Complete=> ,(*mapped in cell services*)
					(*The following are for Binzel type reamers only*)
					LifterUp_ACK=> , (*mapped in cell services*)
					Clamp_ACK=>,(*mapped in cell services*)
					Injector_ACK=> ,(*mapped in cell services*)
					WireCutter_ACK=> (*mapped in cell services*)
					);
			(*R8.Reamer[1](
				(*FB Inputs*)
					Enable_Motion:= All_Estops_OK,
					Fronius_Ream:= TRUE,
                    Binzel_Ream:= FALSE,  (*optional*)
					Ream_REQ:= R8.Peripheral_Req.5 AND (R8.Task_ID_Ack=Tip_Dress),

				(*FB Outputs*)
					Reaming_Complete=> ,(*mapped in cell services*)
					);*)
		(*Call Actual Object*)
		R8();
		(*Output Data*)
		Out_To_ICxx.Robot[8].Robot_Type:= R8.FB_In.Robot_Type;
		Out_To_ICxx.Robot[8].Status:= R8.Status;
		Out_To_ICxx.Robot[8].Axis_Data[1]:= R8.S_Axis_Pos_Raw;
		Out_To_ICxx.Robot[8].In_Image:= R8.Input_Image;
		Out_To_ICxx.Robot[8].Out_Image:= R8.Output_Image;
		Out_To_ICxx.Robot[8].Discrete_ImageFSOE:= R8.Discrete_Image_FSoE;
		Out_To_ICxx.Robot[8].Options:= R8.FB_In.Options;
			Out_To_ICxx.Robot[8].WS_Discrete_Image[1]:= R8.WS[1].Discrete_Image;
			Out_To_ICxx.Robot[8].WS_Discrete_Image[2]:= R8.WS[2].Discrete_Image;
 			Out_To_ICxx.Robot[8].ATI_Discrete_Image:= R8.ATI[1].Discrete_Image;
			Out_To_ICxx.Robot[8].Reamer_Discrete_Image:= R8.Reamer[1].Discrete_Image;
			Out_To_ICxx.Robot[8].Fronius_Status:= R8.Fronius_Status;
		Out_To_ICxx.Robot[8].Ped_IO_ToShow[1]:= 0;			(*Set to Ped value if this robots ecat string contains the Ped's IO*)
		Out_To_ICxx.Robot[8].Ped_IO_ToShow[2]:= 0;			(*Set to Ped value if this robots ecat string contains the Ped's IO*)
		Out_To_ICxx.Robot[8].ECAT_Cable_Breaks:= R8.ECatSlave_Cable_Breaks;
		Out_To_ICxx.Robot[8].CT:= R8.CT;



(*R9 ------------------------*)
		(*Input Data*)
		R9.FB_In.Robot_Type:=KUKA_KRC4_SAFEOP;
		R9.FB_In.Install_Zero_Orientation:= 0; 	(*Set this value between 0 and 359 to set the zero position of the robot physical install with reference to 12 o'clock symbol on UI screens*)
		R9.FB_In.Under_Construction:= GTAC_CONFIG.Under_Construction;
		R9.FB_In.In_SIM_Mode:= GTAC_CONFIG.In_SIM_Mode;
		R9.FB_In.SIM_StartWorkAround:= FALSE;  (*Main.SIM_WorkAround_StartRobots*)
		R9.FB_In.CoE_Read_Trigger:= (GTAC_CONFIG.Option_Robot_Count>=9) AND Pulse_CoERead;
		R9.FB_In.Ecat_Master_AmsNetID:= MAIN.ECAT_Master.AmsID;
		R9.FB_In.Prev_EcatNode_Present:= NOT R8.EK1100_NotPresent; (*Ensure Previous Node Exists to determine Ecat Cable Break of this Devices Input Cable*)
		R9.FB_In.Safety_RST:=SAFETY_RESET;
		R9.FB_In.Enable_Motion:= All_Estops_OK OR GTAC_CONFIG.Under_Construction;
		R9.FB_In.Alarm_RST:=In_From_ICxx.ControlPower1;
		R9.FB_In.Select_Play:=FALSE;
		R9.FB_In.Select_Teach:=FALSE;
		R9.FB_In.Select_Remote:=FALSE;
		R9.FB_In.Start_Scan:=In_From_ICxx.StartRobots;
		R9.FB_In.Stop_Scan:=In_From_ICxx.StopRobots;
		R9.FB_In.Stop_Scan2:=FALSE;
		R9.FB_In.In_DryCycle:= GTAC_CONFIG.Dry_Cycle_Enabled;
		R9.FB_In.Low_Speed:= GTAC_CONFIG.Low_Speed_Enabled;
		R9.FB_In.Speed_Request:= In_From_ICxx.Global_Robot_Speed;
		R9.FB_In.Force_MasterTest_Req:= Cell_Services_Prog.Human_Reqs_MasterTest OR Cell_Services_Prog.A_Robot_Reqs_MasterTest;
		R9.FB_In.Force_BrakeTest_Req:= Cell_Services_Prog.Human_Reqs_BrakeTest OR Cell_Services_Prog.A_Robot_Reqs_BrakeTest;
		R9.FB_In.Major_Faults:= Faults.System_Major_Fault;
		R9.FB_In.Teach_Interlock:=R9_Data.Teach_Interlock;
		R9.FB_In.Weld_Inhibit:=In_From_ICxx.Rxx_Weld_Inhibit;
		R9.FB_In.Option_Disable_WaterFLT:= FALSE AND GTAC_CONFIG.Under_Construction OR (MAIN.R9.Task_ID_Ack=Tip_Change_EXT); (*Used to disable water fault if no water is present. use with caution*)
		R9.FB_In.OK_ToEnter_EquipInterf1:=R9_Data.OK_ToEnter_EquipInterf1;
		R9.FB_In.OK_ToEnter_EquipInterf2:=R9_Data.OK_ToEnter_EquipInterf2;
		R9.FB_In.OK_ToEnter_EquipInterf3:=R9_Data.OK_ToEnter_EquipInterf3;
		R9.FB_In.OK_ToEnter_EquipInterf4:=R9_Data.OK_ToEnter_EquipInterf4;
		R9.FB_In.OK_ToEnter_EquipInterf5:=R9_Data.OK_ToEnter_EquipInterf5;
		R9.FB_In.OK_ToEnter_EquipInterf6:=R9_Data.OK_ToEnter_EquipInterf6;
		R9.FB_In.OK_ToEnter_EquipInterf7:=R9_Data.OK_ToEnter_EquipInterf7;
		R9.FB_In.OK_ToEnter_EquipInterf8:=R9_Data.OK_ToEnter_EquipInterf8;
		R9.FB_In.OK_ToEnter_EquipInterf9:=R9_Data.OK_ToEnter_EquipInterf9;
		R9.FB_In.OK_ToEnter_HumanInterf1:=R9_Data.OK_ToEnter_HumanInterf1;
		R9.FB_In.OK_ToEnter_HumanInterf2:=R9_Data.OK_ToEnter_HumanInterf2;
		R9.FB_In.OK_ToEnter_HumanInterf3:=R9_Data.OK_ToEnter_HumanInterf3;
		R9.FB_In.OK_ToEnter_HumanInterf4:=R9_Data.OK_ToEnter_HumanInterf4;
		R9.FB_In.OK_ToEnter_HumanInterf5:=R9_Data.OK_ToEnter_HumanInterf5;
		R9.FB_In.OK_ToEnter_HumanInterf6:=R9_Data.OK_ToEnter_HumanInterf6;
		R9.FB_In.OK_ToEnter_HumanInterf7:=R9_Data.OK_ToEnter_HumanInterf7;
		R9.FB_In.OK_ToEnter_HumanInterf8:=R9_Data.OK_ToEnter_HumanInterf8;
		R9.FB_In.OK_ToEnter_RobotInterfs:= R9_Data.OK_ToEnter_RobotInterfs;
		R9.FB_In.Fix_ID:=R9_Data.Fix_ID[R9.Location_Index];
		R9.FB_In.Model_ID:=R9_Data.Model_ID[R9.Location_Index];
		R9.FB_In.Task_ID:=R9_Data.Task_ID[R9.Location_Index];
		R9.FB_In.Proceed_From_Pounce:=R9_Data.Proceed_From_Pounce[R9.Location_Index];
		R9.FB_In.Complete_Ack:=R9_Data.Complete_Ack[R9.Location_Index];
		R9.FB_In.PeripheralReq_Ack:=R9_Data.PeripheralReq_Ack[R9.Location_Index];
		R9.FB_In.AuxReq_Ack:=R9_Data.AuxReq_Ack[R9.Location_Index];
		R9.FB_In.User_Inputs.0:= FALSE;
		R9.FB_In.User_Inputs.1:= FALSE;
		R9.FB_In.User_Inputs.2:= FALSE;
		R9.FB_In.User_Inputs.3:= FALSE;
		R9.FB_In.User_Inputs.4:= FALSE;
		R9.FB_In.User_Inputs.5:= FALSE;
		R9.FB_In.User_Inputs.6:= FALSE;
		R9.FB_In.User_Inputs.7:= FALSE;
			(*Configure Options Amounts*)
			R9.FB_In.Options.WeldCont_Amount:= 0; 					(*Select amount of Spot Type Weld Controllers here (0 min, 4 max)*)
			R9.FB_In.Options.WaterStand_Amount:= 0;				(*Select amount of Water Stands here (0 min, 2 max)*)
			R9.FB_In.Options.MIGCont_Amount:= 1;					(*Select amount of MIG Type Weld Controllers here (0 min, 1 max)*)
			R9.FB_In.Options.Reamer_Amount:= 1;					(*Select amount of Tip Reamers here (0 min, 1 max)*)
			R9.FB_In.Options.EOAT_Amount:= 0;						(*Assign EOAT number to robot (0 min, 10 max)*)
			(*Configure Options Parameters*)
			
			R9.Reamer[1](
				(*FB Inputs*)
					Enable_Motion:= All_Estops_OK,
					Fronius_Ream:= TRUE,
                    Binzel_Ream:= FALSE,  (*optional*)
					
					Ream_REQ:= R9.Peripheral_Req.1 AND ((R9.Task_ID_Ack=Tip_Dress)OR (R9.In_T1 AND R9.Peripheral_Req.5)),
					Ream_Time:= T#2S,
					Ream_Clamp_Open:= R9.Reamer[1].N01.I.1,
					Spray_REQ:= R9.Peripheral_Req.2 AND ((R9.Task_ID_Ack=Tip_Dress)OR (R9.In_T1 AND R9.Peripheral_Req.5)),
					Spray_Time:= T#2S,
					F_WireCutter_REQ:= R9.Peripheral_Req.4 AND ((R9.Task_ID_Ack=Tip_Dress)OR (R9.In_T1 AND R9.Peripheral_Req.5)),
					F_WireCutter_Time:= T#1S,
					
				(*FB Outputs*)
					Reaming_Complete=> ,(*mapped in cell services*)
					(*The following are for Binzel type reamers only*)
					LifterUp_ACK=> , (*mapped in cell services*)
					Clamp_ACK=>,(*mapped in cell services*)
					Injector_ACK=> ,(*mapped in cell services*)
					WireCutter_ACK=> (*mapped in cell services*)
					);
			(*R9.Reamer[1](
				(*FB Inputs*)
					Enable_Motion:= All_Estops_OK,
					Fronius_Ream:= TRUE,
                    Binzel_Ream:= FALSE,  (*optional*)
					Ream_REQ:= R9.Peripheral_Req.5 AND (R9.Task_ID_Ack=Tip_Dress),

				(*FB Outputs*)
					Reaming_Complete=> ,(*mapped in cell services*)
					);*)
		(*Call Actual Object*)
		R9();
		(*Output Data*)
		Out_To_ICxx.Robot[9].Robot_Type:= R9.FB_In.Robot_Type;
		Out_To_ICxx.Robot[9].Status:= R9.Status;
		Out_To_ICxx.Robot[9].Axis_Data[1]:= R9.S_Axis_Pos_Raw;
		Out_To_ICxx.Robot[9].In_Image:= R9.Input_Image;
		Out_To_ICxx.Robot[9].Out_Image:= R9.Output_Image;
		Out_To_ICxx.Robot[9].Discrete_ImageFSOE:= R9.Discrete_Image_FSoE;
		Out_To_ICxx.Robot[9].Options:= R9.FB_In.Options;
			Out_To_ICxx.Robot[9].WS_Discrete_Image[1]:= R9.WS[1].Discrete_Image;
			Out_To_ICxx.Robot[9].WS_Discrete_Image[2]:= R9.WS[2].Discrete_Image;
 			Out_To_ICxx.Robot[9].ATI_Discrete_Image:= R9.ATI[1].Discrete_Image;
			Out_To_ICxx.Robot[9].Reamer_Discrete_Image:= R9.Reamer[1].Discrete_Image;
			Out_To_ICxx.Robot[9].Fronius_Status:= R9.Fronius_Status;
		Out_To_ICxx.Robot[9].Ped_IO_ToShow[1]:= 0;			(*Set to Ped value if this robots ecat string contains the Ped's IO*)
		Out_To_ICxx.Robot[9].Ped_IO_ToShow[2]:= 0;			(*Set to Ped value if this robots ecat string contains the Ped's IO*)
		Out_To_ICxx.Robot[9].ECAT_Cable_Breaks:= R9.ECatSlave_Cable_Breaks;
		Out_To_ICxx.Robot[9].CT:= R9.CT;



(*R10 ------------------------*)
		(*Input Data*)
		R10.FB_In.Robot_Type:=KUKA_KRC4_SAFEOP;
		R10.FB_In.Install_Zero_Orientation:= 0; 	(*Set this value between 0 and 359 to set the zero position of the robot physical install with reference to 12 o'clock symbol on UI screens*)
		R10.FB_In.Under_Construction:= GTAC_CONFIG.Under_Construction;
		R10.FB_In.In_SIM_Mode:= GTAC_CONFIG.In_SIM_Mode;
		R10.FB_In.SIM_StartWorkAround:= FALSE;  (*Main.SIM_WorkAround_StartRobots*)
		R10.FB_In.CoE_Read_Trigger:= (GTAC_CONFIG.Option_Robot_Count>=10) AND Pulse_CoERead;
		R10.FB_In.Ecat_Master_AmsNetID:= MAIN.ECAT_Master.AmsID;
		R10.FB_In.Prev_EcatNode_Present:= NOT R9.EK1100_NotPresent; (*Ensure Previous Node Exists to determine Ecat Cable Break of this Devices Input Cable*)
		R10.FB_In.Safety_RST:=SAFETY_RESET;
		R10.FB_In.Enable_Motion:= All_Estops_OK OR GTAC_CONFIG.Under_Construction;
		R10.FB_In.Alarm_RST:=In_From_ICxx.ControlPower1;
		R10.FB_In.Select_Play:=FALSE;
		R10.FB_In.Select_Teach:=FALSE;
		R10.FB_In.Select_Remote:=FALSE;
		R10.FB_In.Start_Scan:=In_From_ICxx.StartRobots;
		R10.FB_In.Stop_Scan:=In_From_ICxx.StopRobots;
		R10.FB_In.Stop_Scan2:=FALSE;
		R10.FB_In.In_DryCycle:= GTAC_CONFIG.Dry_Cycle_Enabled;
		R10.FB_In.Low_Speed:= GTAC_CONFIG.Low_Speed_Enabled;
		R10.FB_In.Speed_Request:= In_From_ICxx.Global_Robot_Speed;
		R10.FB_In.Force_MasterTest_Req:= Cell_Services_Prog.Human_Reqs_MasterTest OR Cell_Services_Prog.A_Robot_Reqs_MasterTest;
		R10.FB_In.Force_BrakeTest_Req:= Cell_Services_Prog.Human_Reqs_BrakeTest OR Cell_Services_Prog.A_Robot_Reqs_BrakeTest;
		R10.FB_In.Major_Faults:= Faults.System_Major_Fault;
		R10.FB_In.Teach_Interlock:=R10_Data.Teach_Interlock;
		R10.FB_In.Weld_Inhibit:=In_From_ICxx.Rxx_Weld_Inhibit;
		R10.FB_In.Option_Disable_WaterFLT:= FALSE AND GTAC_CONFIG.Under_Construction OR (MAIN.R10.Task_ID_Ack=Tip_Change_EXT); (*Used to disable water fault if no water is present. use with caution*)
		R10.FB_In.OK_ToEnter_EquipInterf1:=R10_Data.OK_ToEnter_EquipInterf1;
		R10.FB_In.OK_ToEnter_EquipInterf2:=R10_Data.OK_ToEnter_EquipInterf2;
		R10.FB_In.OK_ToEnter_EquipInterf3:=R10_Data.OK_ToEnter_EquipInterf3;
		R10.FB_In.OK_ToEnter_EquipInterf4:=R10_Data.OK_ToEnter_EquipInterf4;
		R10.FB_In.OK_ToEnter_EquipInterf5:=R10_Data.OK_ToEnter_EquipInterf5;
		R10.FB_In.OK_ToEnter_EquipInterf6:=R10_Data.OK_ToEnter_EquipInterf6;
		R10.FB_In.OK_ToEnter_EquipInterf7:=R10_Data.OK_ToEnter_EquipInterf7;
		R10.FB_In.OK_ToEnter_EquipInterf8:=R10_Data.OK_ToEnter_EquipInterf8;
		R10.FB_In.OK_ToEnter_EquipInterf9:=R10_Data.OK_ToEnter_EquipInterf9;
		R10.FB_In.OK_ToEnter_HumanInterf1:=R10_Data.OK_ToEnter_HumanInterf1;
		R10.FB_In.OK_ToEnter_HumanInterf2:=R10_Data.OK_ToEnter_HumanInterf2;
		R10.FB_In.OK_ToEnter_HumanInterf3:=R10_Data.OK_ToEnter_HumanInterf3;
		R10.FB_In.OK_ToEnter_HumanInterf4:=R10_Data.OK_ToEnter_HumanInterf4;
		R10.FB_In.OK_ToEnter_HumanInterf5:=R10_Data.OK_ToEnter_HumanInterf5;
		R10.FB_In.OK_ToEnter_HumanInterf6:=R10_Data.OK_ToEnter_HumanInterf6;
		R10.FB_In.OK_ToEnter_HumanInterf7:=R10_Data.OK_ToEnter_HumanInterf7;
		R10.FB_In.OK_ToEnter_HumanInterf8:=R10_Data.OK_ToEnter_HumanInterf8;
		R10.FB_In.OK_ToEnter_RobotInterfs:= R10_Data.OK_ToEnter_RobotInterfs;
		R10.FB_In.Fix_ID:=R10_Data.Fix_ID[R10.Location_Index];
		R10.FB_In.Model_ID:=R10_Data.Model_ID[R10.Location_Index];
		R10.FB_In.Task_ID:=R10_Data.Task_ID[R10.Location_Index];
		R10.FB_In.Proceed_From_Pounce:=R10_Data.Proceed_From_Pounce[R10.Location_Index];
		R10.FB_In.Complete_Ack:=R10_Data.Complete_Ack[R10.Location_Index];
		R10.FB_In.PeripheralReq_Ack:=R10_Data.PeripheralReq_Ack[R10.Location_Index];
		R10.FB_In.AuxReq_Ack:=R10_Data.AuxReq_Ack[R10.Location_Index];
		R10.FB_In.User_Inputs.0:= FALSE;
		R10.FB_In.User_Inputs.1:= FALSE;
		R10.FB_In.User_Inputs.2:= FALSE;
		R10.FB_In.User_Inputs.3:= FALSE;
		R10.FB_In.User_Inputs.4:= FALSE;
		R10.FB_In.User_Inputs.5:= FALSE;
		R10.FB_In.User_Inputs.6:= FALSE;
		R10.FB_In.User_Inputs.7:= FALSE;
			(*Configure Options Amounts*)
			R10.FB_In.Options.WeldCont_Amount:= 0; 					(*Select amount of Spot Type Weld Controllers here (0 min, 4 max)*)
			R10.FB_In.Options.WaterStand_Amount:= 0;				(*Select amount of Water Stands here (0 min, 2 max)*)
			R10.FB_In.Options.MIGCont_Amount:= 1;					(*Select amount of MIG Type Weld Controllers here (0 min, 1 max)*)
			R10.FB_In.Options.Reamer_Amount:= 1;					(*Select amount of Tip Reamers here (0 min, 1 max)*)
			R10.FB_In.Options.EOAT_Amount:= 0;					(*Assign EOAT number to robot (0 min, 10 max)*)
			(*Configure Options Parameters*)
			(*R10.Reamer[1](
				(*FB Inputs*)
					Enable_Motion:= All_Estops_OK,
					Fronius_Ream:= TRUE,
                    Binzel_Ream:= FALSE,  (*optional*)
					Ream_REQ:= R10.Peripheral_Req.5 AND (R10.Task_ID_Ack=Tip_Dress),

				(*FB Outputs*)
					Reaming_Complete=> ,(*mapped in cell services*)
					);*)
		(*Call Actual Object*)
		R10();
		(*Output Data*)
		Out_To_ICxx.Robot[10].Robot_Type:= R10.FB_In.Robot_Type;
		(*To create less work, since there is no welding, changeing this number to 307 so we dont have to mess with the kuka FB, just screens. "us_Rxx_Status" - added 307 "inspecting"*)
		IF (R10.Status = 305) THEN
		Out_To_ICxx.Robot[10].Status:= 307; 
		ELSE
		Out_To_ICxx.Robot[10].Status:= R10.Status;
		END_IF
		Out_To_ICxx.Robot[10].Axis_Data[1]:= R10.S_Axis_Pos_Raw;
		Out_To_ICxx.Robot[10].In_Image:= R10.Input_Image;
		Out_To_ICxx.Robot[10].Out_Image:= R10.Output_Image;
		Out_To_ICxx.Robot[10].Discrete_ImageFSOE:= R10.Discrete_Image_FSoE;
		Out_To_ICxx.Robot[10].Options:= R10.FB_In.Options;
			Out_To_ICxx.Robot[10].WS_Discrete_Image[1]:= R10.WS[1].Discrete_Image;
			Out_To_ICxx.Robot[10].WS_Discrete_Image[2]:= R10.WS[2].Discrete_Image;
 			Out_To_ICxx.Robot[10].ATI_Discrete_Image:= R10.ATI[1].Discrete_Image;
			Out_To_ICxx.Robot[10].Reamer_Discrete_Image:= R10.Reamer[1].Discrete_Image;
			Out_To_ICxx.Robot[10].Fronius_Status:= R10.Fronius_Status;
		Out_To_ICxx.Robot[10].Ped_IO_ToShow[1]:= 0;			(*Set to Ped value if this robots ecat string contains the Ped's IO*)
		Out_To_ICxx.Robot[10].Ped_IO_ToShow[2]:= 0;			(*Set to Ped value if this robots ecat string contains the Ped's IO*)
		Out_To_ICxx.Robot[10].ECAT_Cable_Breaks:= R10.ECatSlave_Cable_Breaks;
		Out_To_ICxx.Robot[10].CT:= R10.CT;



(*R11 ------------------------*)
		(*Input Data*)
		R11.FB_In.Robot_Type:=KUKA_KRC4_SAFEOP;
		R11.FB_In.Install_Zero_Orientation:= 0; 	(*Set this value between 0 and 359 to set the zero position of the robot physical install with reference to 12 o'clock symbol on UI screens*)
		R11.FB_In.Under_Construction:= GTAC_CONFIG.Under_Construction;
		R11.FB_In.In_SIM_Mode:= GTAC_CONFIG.In_SIM_Mode;
		R11.FB_In.SIM_StartWorkAround:= FALSE;  (*Main.SIM_WorkAround_StartRobots*)
		R11.FB_In.CoE_Read_Trigger:= (GTAC_CONFIG.Option_Robot_Count>=11) AND Pulse_CoERead;
		R11.FB_In.Ecat_Master_AmsNetID:= MAIN.ECAT_Master.AmsID;
		R11.FB_In.Prev_EcatNode_Present:= NOT R10.EK1100_NotPresent; (*Ensure Previous Node Exists to determine Ecat Cable Break of this Devices Input Cable*)
		R11.FB_In.Safety_RST:=SAFETY_RESET;
		R11.FB_In.Enable_Motion:= All_Estops_OK OR GTAC_CONFIG.Under_Construction;
		R11.FB_In.Alarm_RST:=In_From_ICxx.ControlPower1;
		R11.FB_In.Select_Play:=FALSE;
		R11.FB_In.Select_Teach:=FALSE;
		R11.FB_In.Select_Remote:=FALSE;
		R11.FB_In.Start_Scan:=In_From_ICxx.StartRobots;
		R11.FB_In.Stop_Scan:=In_From_ICxx.StopRobots;
		R11.FB_In.Stop_Scan2:=FALSE;
		R11.FB_In.In_DryCycle:= GTAC_CONFIG.Dry_Cycle_Enabled;
		R11.FB_In.Low_Speed:= GTAC_CONFIG.Low_Speed_Enabled;
		R11.FB_In.Speed_Request:= In_From_ICxx.Global_Robot_Speed;
		R11.FB_In.Force_MasterTest_Req:= Cell_Services_Prog.Human_Reqs_MasterTest OR Cell_Services_Prog.A_Robot_Reqs_MasterTest;
		R11.FB_In.Force_BrakeTest_Req:= Cell_Services_Prog.Human_Reqs_BrakeTest OR Cell_Services_Prog.A_Robot_Reqs_BrakeTest;
		R11.FB_In.Major_Faults:= Faults.System_Major_Fault;
		R11.FB_In.Teach_Interlock:=R11_Data.Teach_Interlock;
		R11.FB_In.Weld_Inhibit:=In_From_ICxx.Rxx_Weld_Inhibit;
		R11.FB_In.Option_Disable_WaterFLT:= FALSE AND GTAC_CONFIG.Under_Construction OR (MAIN.R11.Task_ID_Ack=Tip_Change_EXT); (*Used to disable water fault if no water is present. use with caution*)
		R11.FB_In.OK_ToEnter_EquipInterf1:=R11_Data.OK_ToEnter_EquipInterf1;
		R11.FB_In.OK_ToEnter_EquipInterf2:=R11_Data.OK_ToEnter_EquipInterf2;
		R11.FB_In.OK_ToEnter_EquipInterf3:=R11_Data.OK_ToEnter_EquipInterf3;
		R11.FB_In.OK_ToEnter_EquipInterf4:=R11_Data.OK_ToEnter_EquipInterf4;
		R11.FB_In.OK_ToEnter_EquipInterf5:=R11_Data.OK_ToEnter_EquipInterf5;
		R11.FB_In.OK_ToEnter_EquipInterf6:=R11_Data.OK_ToEnter_EquipInterf6;
		R11.FB_In.OK_ToEnter_EquipInterf7:=R11_Data.OK_ToEnter_EquipInterf7;
		R11.FB_In.OK_ToEnter_EquipInterf8:=R11_Data.OK_ToEnter_EquipInterf8;
		R11.FB_In.OK_ToEnter_EquipInterf9:=R11_Data.OK_ToEnter_EquipInterf9;
		R11.FB_In.OK_ToEnter_HumanInterf1:=R11_Data.OK_ToEnter_HumanInterf1;
		R11.FB_In.OK_ToEnter_HumanInterf2:=R11_Data.OK_ToEnter_HumanInterf2;
		R11.FB_In.OK_ToEnter_HumanInterf3:=R11_Data.OK_ToEnter_HumanInterf3;
		R11.FB_In.OK_ToEnter_HumanInterf4:=R11_Data.OK_ToEnter_HumanInterf4;
		R11.FB_In.OK_ToEnter_HumanInterf5:=R11_Data.OK_ToEnter_HumanInterf5;
		R11.FB_In.OK_ToEnter_HumanInterf6:=R11_Data.OK_ToEnter_HumanInterf6;
		R11.FB_In.OK_ToEnter_HumanInterf7:=R11_Data.OK_ToEnter_HumanInterf7;
		R11.FB_In.OK_ToEnter_HumanInterf8:=R11_Data.OK_ToEnter_HumanInterf8;
		R11.FB_In.OK_ToEnter_RobotInterfs:= R11_Data.OK_ToEnter_RobotInterfs;
		R11.FB_In.Fix_ID:=R11_Data.Fix_ID[R11.Location_Index];
		R11.FB_In.Model_ID:=R11_Data.Model_ID[R11.Location_Index];
		R11.FB_In.Task_ID:=R11_Data.Task_ID[R11.Location_Index];
		R11.FB_In.Proceed_From_Pounce:=R11_Data.Proceed_From_Pounce[R11.Location_Index];
		R11.FB_In.Complete_Ack:=R11_Data.Complete_Ack[R11.Location_Index];
		R11.FB_In.PeripheralReq_Ack:=R11_Data.PeripheralReq_Ack[R11.Location_Index];
		R11.FB_In.AuxReq_Ack:=R11_Data.AuxReq_Ack[R11.Location_Index];
		R11.FB_In.User_Inputs.0:= FALSE;
		R11.FB_In.User_Inputs.1:= FALSE;
		R11.FB_In.User_Inputs.2:= FALSE;
		R11.FB_In.User_Inputs.3:= FALSE;
		R11.FB_In.User_Inputs.4:= FALSE;
		R11.FB_In.User_Inputs.5:= FALSE;
		R11.FB_In.User_Inputs.6:= FALSE;
		R11.FB_In.User_Inputs.7:= FALSE;
			(*Configure Options Amounts*)
			R11.FB_In.Options.WeldCont_Amount:= 0; 					(*Select amount of Spot Type Weld Controllers here (0 min, 4 max)*)
			R11.FB_In.Options.WaterStand_Amount:= 0;				(*Select amount of Water Stands here (0 min, 2 max)*)
			R11.FB_In.Options.MIGCont_Amount:= 1;					(*Select amount of MIG Type Weld Controllers here (0 min, 1 max)*)
			R11.FB_In.Options.Reamer_Amount:= 1;					(*Select amount of Tip Reamers here (0 min, 1 max)*)
			R11.FB_In.Options.EOAT_Amount:= 0;					(*Assign EOAT number to robot (0 min, 10 max)*)
			(*Configure Options Parameters*)
			(*R11.Reamer[1](
				(*FB Inputs*)
					Enable_Motion:= All_Estops_OK,
					Fronius_Ream:= TRUE,
                    Binzel_Ream:= FALSE,  (*optional*)
					Ream_REQ:= R11.Peripheral_Req.5 AND (R11.Task_ID_Ack=Tip_Dress),

				(*FB Outputs*)
					Reaming_Complete=> ,(*mapped in cell services*)
					);*)
		(*Call Actual Object*)
		R11();
		(*Output Data*)
		Out_To_ICxx.Robot[11].Robot_Type:= R11.FB_In.Robot_Type;
		(*To create less work, since there is no welding, changeing this number to 307 so we dont have to mess with the kuka FB, just screens. "us_Rxx_Status" - added 307 "inspecting"*)
		IF (R11.Status = 305) THEN
		Out_To_ICxx.Robot[11].Status:= 307; 
		ELSE
		Out_To_ICxx.Robot[11].Status:= R11.Status;
		END_IF
		Out_To_ICxx.Robot[11].Axis_Data[1]:= R11.S_Axis_Pos_Raw;
		Out_To_ICxx.Robot[11].In_Image:= R11.Input_Image;
		Out_To_ICxx.Robot[11].Out_Image:= R11.Output_Image;
		Out_To_ICxx.Robot[11].Discrete_ImageFSOE:= R11.Discrete_Image_FSoE;
		Out_To_ICxx.Robot[11].Options:= R11.FB_In.Options;
			Out_To_ICxx.Robot[11].WS_Discrete_Image[1]:= R11.WS[1].Discrete_Image;
			Out_To_ICxx.Robot[11].WS_Discrete_Image[2]:= R11.WS[2].Discrete_Image;
 			Out_To_ICxx.Robot[11].ATI_Discrete_Image:= R11.ATI[1].Discrete_Image;
			Out_To_ICxx.Robot[11].Reamer_Discrete_Image:= R11.Reamer[1].Discrete_Image;
			Out_To_ICxx.Robot[11].Fronius_Status:= R11.Fronius_Status;
		Out_To_ICxx.Robot[11].Ped_IO_ToShow[1]:= 0;			(*Set to Ped value if this robots ecat string contains the Ped's IO*)
		Out_To_ICxx.Robot[11].Ped_IO_ToShow[2]:= 0;			(*Set to Ped value if this robots ecat string contains the Ped's IO*)
		Out_To_ICxx.Robot[11].ECAT_Cable_Breaks:= R11.ECatSlave_Cable_Breaks;
		Out_To_ICxx.Robot[11].CT:= R11.CT;























(*end*)
END_ACTION

(* stored: Version 1.1.0.1, ProductVersion 3.1.4024.12
   POU MAIN: Id {84c1c1eb-535c-4ffe-828a-2356a4a2ae04}, SpecialFunc None
   Action EOATs: Id {74536ccf-3a76-4949-acf9-11e995ae86cc}
   Action ICs: Id {deccbd85-5f42-4b64-8e81-375e56a63756}
   Action Product_Tracking: Id {b180e8a1-2952-497b-b976-b2c524bb6089}
   Action Robots: Id {24524792-0aca-4eae-af81-38966ec4ed01} *)
